{attribute 'GeneratedUsingTerminal: EP9576-1032-0016'}
{attribute addProperty BoxType "EP9576-1032-0016"}
{attribute addProperty Id "BCT_InputsAT %I*BCT_Inputs_7ACE8FA617WcStateAT %I*WcState_9091E0EB2InfoDataAT %I*InfoData_94A18F5E2"}
{attribute addProperty CRC "4086821292"}
{attribute addProperty Size "21"}
TYPE EP9576_F397F1AC EXTENDS EtcSlaveTerminalBase_947E5A46 :
STRUCT
	{attribute addProperty Name "BCT_Inputs"}
	BCT_Inputs : BCT_Inputs_7ACE8FA6;
	{attribute addProperty Name "WcState"}
	WcState : WcState_9091E0EB;
	{attribute addProperty Name "InfoData"}
	InfoData : InfoData_94A18F5E;
END_STRUCT
END_TYPE

(* stored: Version 1.2.0.0, ProductVersion 3.1.4024.9
   DUT EP9576_F397F1AC: Id {c6b11c24-2c43-4022-a3de-d11b255333af} *)
